Universal Robots PolyScope program: Step Corner Left Around.urp

Program Step Corner Left Around (installation=default directory=/programs createdIn=5.21.3 lastSavedIn=5.21.3 robotSerialNumber=20246801938)
Calibrated DH parameters: a=[-0.000071, -0.790281, -0.600694, 0.000061, -0.000039, 0]; d=[0.236272, 604.465945, 132.116513, -736.382239, 0.159268, 0.154005]; alpha=[1.570254, -0.000567, 0.000559, 1.571709, -1.56999, 0]; deltaTheta=[0, -0.409357, 7.293326, -0.600784, -0.000001, -0.000001]
InitVariablesNode
Robot Program (runOnlyOnce=false)
  Folder dummy points
    MoveJ speed 60 deg/s, acceleration 80 deg/s^2 (useActiveTCP=true optimoveEnabled=false optiMoveSpeed=0.3 optiMoveAcceleration=0.09) feature=Base
      Waypoint Waypoint_1: TCP in base x=-1359.076 y=96.899 z=76.714 mm, rx=-1.5536 ry=-0.3564 rz=0.3809 rad; joints [4.419, -22.046, 46.907, -25.955, -112.41, 88.981] deg; TCP offset x=-9.5 y=-328 z=105.73 mm, rx=1.2092 ry=-1.2092 rz=1.2092 rad
      Waypoint Waypoint_2: TCP in base x=-1360.87 y=94.224 z=-76.422 mm, rx=-1.5536 ry=-0.3564 rz=0.3809 rad; joints [4.515, -15.342, 45.323, -31.071, -112.316, 88.988] deg
